FUNCTION_BLOCK SKILL_Param_BOOL (* Skill parameter (BOOL): default, range check of a Start argument, latching for one run *)
  (* Standard: 61499-2 *)
  (* Version 0.1, 2026-09-28, Project contributors, AAU Smart Production Lab *)
  PACKAGE modlib;
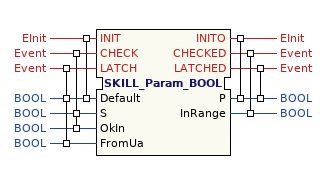
  EVENT_INPUT
    INIT : EInit WITH Default;
    CHECK WITH S, OkIn;
    LATCH WITH FromUa, Default;
  END_EVENT
  EVENT_OUTPUT
    INITO : EInit WITH P;
    CHECKED WITH InRange;
    LATCHED WITH P;
  END_EVENT
  VAR_INPUT
    Default : BOOL;
    S : BOOL;
    OkIn : BOOL := TRUE;
    FromUa : BOOL;
  END_VAR
  VAR_OUTPUT
    P : BOOL;
    InRange : BOOL;
  END_VAR
  EC_STATES
    INIT : INIT -> INITO;
    CHECK : CHECK -> CHECKED;
    LATCH : LATCH -> LATCHED;
  END_STATES
  ALGORITHM INIT IN ST:
P := Default;
  END_ALGORITHM
  ALGORITHM CHECK IN ST:
InRange := OkIn;
  END_ALGORITHM
  ALGORITHM LATCH IN ST:
IF FromUa THEN
  P := S;
ELSE
  P := Default;
END_IF;
  END_ALGORITHM
END_FUNCTION_BLOCK
